// Struckig
// Copyright (C) 2022 Stefan Besler

// This program is free software: you can redistribute it and/or modify
// it under the terms of the GNU General Public License as published by
// the Free Software Foundation, either version 3 of the License, or
// (at your option) any later version.

// This program is distributed in the hope that it will be useful,
// but WITHOUT ANY WARRANTY; without even the implied warranty of
// MERCHANTABILITY or FITNESS FOR A PARTICULAR PURPOSE.  See the
// GNU General Public License for more details.
//
// You should have received a copy of the GNU General Public License
// along with THIS PROGRAM.  IF NOT, see <http://www.gnu.org/licenses/>.
/// Mathematical equations for Step 1 in third-order position interface: Extremal profiles
FUNCTION_BLOCK INTERNAL PositionThirdOrderStep1
VAR
  v0, a0 : LREAL;
  vf, af : LREAL;
  _vMax, _vMin, _aMax, _aMin, _jMax : LREAL;

  // Pre-calculated expressions
  pd : LREAL;
  v0_v0, vf_vf : LREAL;
  a0_a0, a0_p3, a0_p4 : LREAL;
  af_af, af_p3, af_p4 : LREAL;
  jMax_jMax : LREAL;
  
  // runtime  calculated expressions
  polynom_none, polynom_acc0, polynom_acc1 : ARRAY[0..4] OF LREAL;
  orig : LREAL;
  deriv : LREAL;
  t : LREAL;
  i : INT;
  h0, h1, h2, h2_h2, h3, h5, h2_none, h3_acc0, h3_acc1, h0_acc0, h2_acc0, h0_acc1, h2_acc1, q : LREAL;
  t_min, t_max, t_min_none, t_max_none, t_min_acc0, t_max_acc0, t_min_acc1, t_max_acc1 : LREAL;
  t_acc1, t_acc0 : LREAL;
  validProfiles : ARRAY[0..5] OF ProfileDesc; // Max 5 valid profiles + 1 spare for numerical issues
  validProfileCounter : INT := -1;
  
  num_roots_none, num_roots_acc0, num_roots_acc1  : INT;
  roots_none, roots_acc0, roots_acc1 : ARRAY[0..6] OF LREAL;
  roots_none_indices, roots_acc0_indices, roots_acc1_indices : ARRAY[0..6] OF INT;
  left_duration, right_duration : LREAL;   
END_VAR

METHOD AddInterval
VAR_IN_OUT
  interval : BlockInterval;
  Left : ProfileDesc;
  Right : ProfileDesc;
END_VAR
left_duration := Left.t_sum[6] + Left.Brake.Duration + Left.Accel.Duration;
right_duration := Right.t_sum[6] + Right.Brake.Duration + Right.Accel.Duration;
IF (left_duration < right_duration)
THEN
  interval.Left := left_duration;
  interval.Right := right_duration;
  interval.Profile := Right;
  interval.IsUsed := TRUE;
ELSE
  interval.Left := right_duration;
  interval.Right := left_duration;
  interval.Profile := Left;
  interval.IsUsed := TRUE;  
END_IF
END_METHOD

METHOD AddProfile
VAR_IN_OUT CONSTANT
  Profile : ProfileDesc;
END_VAR
validProfileCounter := validProfileCounter + 1;
validProfiles[validProfileCounter] := Profile;
END_METHOD

METHOD CalculateBlock : BOOL
VAR_IN_OUT
  block : Block;
END_VAR
VAR
  i, j : INT;
  Tmin : LREAL;
  idx_min : INT;
  idx_else_1, idx_else_2, idx_else_3, idx_else_4 : INT;
END_VAR
block.A.IsUsed := FALSE;
block.B.IsUsed := FALSE;

IF validProfileCounter = 0
THEN
  block.Pmin := validProfiles[0];
  block.Tmin := block.Pmin.t_sum[6] + block.Pmin.Brake.Duration + block.Pmin.Accel.Duration; 
  CalculateBlock := TRUE;

ELSIF validProfileCounter = 1 
THEN

  IF ABS(validProfiles[0].t_sum[6] - validProfiles[1].t_sum[6]) < 8*Constants.Epsilon
  THEN
    block.Pmin := validProfiles[0];
    block.Tmin := block.Pmin.t_sum[6] + block.Pmin.Brake.Duration + block.Pmin.Accel.Duration;  
    CalculateBlock := TRUE;
    RETURN;
	END_IF
  
  IF ParameterList.NumericalRobust
  THEN
    idx_min := SEL(validProfiles[0].t_sum[6] < validProfiles[1].t_sum[6], 1, 0);
    idx_else_1 := (idx_min + 1) MOD 2;

    block.Pmin := validProfiles[idx_min];
    block.Tmin := block.Pmin.t_sum[6] + block.Pmin.Brake.Duration + block.Pmin.Accel.Duration; 
    AddInterval(block.A, validProfiles[idx_min], validProfiles[idx_else_1]);
    CalculateBlock := TRUE;
    RETURN; 
	END_IF

// Only happens due to numerical issues
ELSIF (validProfileCounter = 3) 
THEN
  // Find "identical" profiles
  IF (ABS(validProfiles[0].t_sum[6] - validProfiles[1].t_sum[6]) < 32*Constants.Epsilon AND_THEN validProfiles[0].Direction <> validProfiles[1].Direction)
  THEN
    RemoveProfile(1);
  ELSIF (ABS(validProfiles[2].t_sum[6] - validProfiles[3].t_sum[6]) < 256*Constants.Epsilon  AND_THEN validProfiles[2].Direction <> validProfiles[3].Direction)
  THEN
    RemoveProfile(3);
  ELSIF (ABS(validProfiles[0].t_sum[6] - validProfiles[3].t_sum[6]) < 256*Constants.Epsilon AND_THEN validProfiles[0].Direction <> validProfiles[3].Direction)
  THEN
    RemoveProfile(3);
  ELSE
    RETURN;
  END_IF

ELSIF ((validProfileCounter+1) MOD 2 = 0)
THEN
  RETURN;
END_IF

// Find index of fastest Profile
Tmin := Constants.Infinity;
FOR i:=0 TO validProfileCounter
DO
  FOR j:=0 TO validProfileCounter
  DO
    IF validProfiles[i].t_sum[6] + validProfiles[i].Brake.Duration < validProfiles[j].t_sum[6] + validProfiles[j].Brake.Duration AND_THEN
       validProfiles[i].t_sum[6] + validProfiles[i].Brake.Duration < Tmin
    THEN
      Tmin := validProfiles[i].t_sum[6] + validProfiles[i].Brake.Duration + validProfiles[i].Accel.Duration;
      idx_min := i;
		END_IF
  END_FOR
END_FOR

block.Pmin := validProfiles[idx_min];
block.Tmin := block.Pmin.t_sum[6] + block.Pmin.Brake.Duration + block.Pmin.Accel.Duration;
IF (validProfileCounter = 2)
THEN
  idx_else_1 := (idx_min + 1) MOD 3;
  idx_else_2 := (idx_min + 2) MOD 3;
  
  AddInterval(block.A, validProfiles[idx_else_1], validProfiles[idx_else_2]);
  CalculateBlock := TRUE;
  RETURN;

 ELSIF (validProfileCounter = 4)
 THEN
  idx_else_1 := (idx_min + 1) MOD 5;
  idx_else_2 := (idx_min + 2) MOD 5;
  idx_else_3 := (idx_min + 3) MOD 5;
  idx_else_4 := (idx_min + 4) MOD 5;
  
  IF (validProfiles[idx_else_1].Direction = validProfiles[idx_else_2].Direction)
  THEN
    AddInterval(block.A, validProfiles[idx_else_1], validProfiles[idx_else_2]);
    AddInterval(block.B, validProfiles[idx_else_3], validProfiles[idx_else_4]);
  ELSE 
    AddInterval(block.A, validProfiles[idx_else_1], validProfiles[idx_else_4]);
    AddInterval(block.B, validProfiles[idx_else_2], validProfiles[idx_else_3]);
  END_IF
  
  CalculateBlock := TRUE;
END_IF
END_METHOD

METHOD Get : BOOL
VAR_INPUT
  input : REFERENCE TO ProfileDesc;
  block : REFERENCE TO Block; 
END_VAR
VAR_INST
  vMax, vMin, aMax, aMin, jMax : LREAL;  
END_VAR
validProfileCounter := -1;

// Zero-limits special case
IF _jMax = 0.0 OR_ELSE _aMax = 0.0 OR_ELSE _aMin = 0.0 
THEN
  block.Pmin.SetBoundary(input);

  IF time_all_single_step(block.Pmin, _vMax, _vMin, _aMax, _aMin, _jMax) 
  THEN
    block.Tmin := block.Pmin.t_sum[6] + block.Pmin.Brake.Duration + block.Pmin.Accel.Duration;
    AddInterval(block.A, block.Pmin, block.Pmin);
    
    IF ABS(v0) > Constants.DoubleEpsilon OR_ELSE ABS(a0) > Constants.DoubleEpsilon
    THEN
	  block.A.Left := block.Tmin;
      block.A.Right := Constants.Infinity;
    END_IF
    
    Get := TRUE;
    RETURN; 
  END_IF
  
  RETURN;
END_IF

validProfiles[0].SetBoundary(input);

IF ABS(vf) < Constants.DoubleEpsilon AND_THEN ABS(af) < Constants.DoubleEpsilon
THEN
  vMax := SEL(pd >= 0, _vMin, _vMax);
  vMin := SEL(pd >= 0, _vMax, _vMin);
  aMax := SEL(pd >= 0, _aMin, _aMax);
  aMin := SEL(pd >= 0, _aMax, _aMin);
  jMax :=SEL (pd >= 0,-_jMax, _jMax);
  
  IF ABS(v0) < Constants.DoubleEpsilon AND_THEN ABS(a0) < Constants.DoubleEpsilon AND_THEN ABS(pd) < Constants.DoubleEpsilon
  THEN
    time_all_none_acc0_acc1(input, vMax, vMin, aMax, aMin, jMax, TRUE);
  ELSE
    // There is no blocked interval when vf==0 && af==0, so return after first found profile
    time_all_vel(input, vMax, vMin, aMax, aMin, jMax, true);
    IF (validProfileCounter >= 0) THEN
      Get := CalculateBlock(block);
      RETURN;
    END_IF
    time_all_none_acc0_acc1(input, vMax, vMin, aMax, aMin, jMax, TRUE);
    IF (validProfileCounter >= 0) THEN
      Get := CalculateBlock(block);
      RETURN;
    END_IF
    time_acc0_acc1(input, vMax, vMin, aMax, aMin, jMax, true);
    IF (validProfileCounter >= 0) THEN
      Get := CalculateBlock(block);
      RETURN;
    END_IF
    
    time_all_vel(input, vMin, vMax, aMin, aMax, -jMax, true);
    IF (validProfileCounter >= 0) THEN
      Get := CalculateBlock(block);
      RETURN;
    END_IF
    time_all_none_acc0_acc1(input, vMin, vMax, aMin, aMax, -jMax, TRUE);
    IF (validProfileCounter >= 0) THEN
      Get := CalculateBlock(block);
      RETURN;
    END_IF
    time_acc0_acc1(input, vMin, vMax, aMin, aMax, -jMax, true);
  END_IF     

ELSE 
  time_all_none_acc0_acc1(input, _vMax, _vMin, _aMax, _aMin, _jMax, FALSE);
  time_all_none_acc0_acc1(input, _vMin, _vMax, _aMin, _aMax, -_jMax, false);
  time_acc0_acc1(input, _vMax, _vMin, _aMax, _aMin, _jMax, false);
  time_acc0_acc1(input, _vMin, _vMax, _aMin, _aMax, -_jMax, FALSE);
  time_all_vel(input, _vMax, _vMin, _aMax, _aMin, _jMax, FALSE);
  time_all_vel(input, _vMin, _vMax, _aMin, _aMax, -_jMax, false);  
END_IF    

IF (validProfileCounter = -1)
THEN
  time_none_two_step(input, _vMax, _vMin, _aMax, _aMin, _jMax);
  IF validProfileCounter >= 0
  THEN
    Get := CalculateBlock(block);
    RETURN;
	END_IF
  
  time_none_two_step(input, _vMin, _vMax, _aMin, _aMax, -_jMax);
  IF validProfileCounter >= 0
  THEN
    Get := CalculateBlock(block);
    RETURN;
	END_IF
  

  time_acc0_two_step(input, _vMax, _vMin, _aMax, _aMin, _jMax);
  IF validProfileCounter >= 0
  THEN
    Get := CalculateBlock(block);
    RETURN;
	END_IF
  
  time_acc0_two_step(input, _vMin, _vMax, _aMin, _aMax, -_jMax);
  IF validProfileCounter >= 0
  THEN
    Get := CalculateBlock(block);
    RETURN;
	END_IF
  
  time_vel_two_step(input, _vMax, _vMin, _aMax, _aMin, _jMax);
  IF validProfileCounter >= 0
  THEN
    Get := CalculateBlock(block);
    RETURN;
	END_IF
  
  time_vel_two_step(input, _vMin, _vMax, _aMin, _aMax, -_jMax);
  IF validProfileCounter >= 0
  THEN
    Get := CalculateBlock(block);
    RETURN;
	END_IF
  
  time_acc1_vel_two_step(input, _vMax, _vMin, _aMax, _aMin, _jMax);
  IF validProfileCounter >= 0
  THEN
    Get := CalculateBlock(block);
    RETURN;
	END_IF
  
  time_acc1_vel_two_step(input, _vMin, _vMax, _aMin, _aMax, -_jMax);
  IF validProfileCounter >= 0
  THEN
    Get := CalculateBlock(block);
    RETURN;
	END_IF  
END_IF

IF (validProfileCounter = -1)
THEN
  time_none_two_step(input, _vMax, _vMin, _aMax, _aMin, _jMax);
  IF validProfileCounter >= 0
  THEN
    Get := CalculateBlock(block);
    RETURN;
	END_IF
  
  time_none_two_step(input, _vMin, _vMax, _aMin, _aMax, -_jMax);
  IF validProfileCounter >= 0
  THEN
    Get := CalculateBlock(block);
    RETURN;
	END_IF
  

  time_acc0_two_step(input, _vMax, _vMin, _aMax, _aMin, _jMax);
  IF validProfileCounter >= 0
  THEN
    Get := CalculateBlock(block);
    RETURN;
	END_IF
  
  time_acc0_two_step(input, _vMin, _vMax, _aMin, _aMax, -_jMax);
  IF validProfileCounter >= 0
  THEN
    Get := CalculateBlock(block);
    RETURN;
	END_IF
  
  time_vel_two_step(input, _vMax, _vMin, _aMax, _aMin, _jMax);
  IF validProfileCounter >= 0
  THEN
    Get := CalculateBlock(block);
    RETURN;
	END_IF
  
  time_vel_two_step(input, _vMin, _vMax, _aMin, _aMax, -_jMax);
  IF validProfileCounter >= 0
  THEN
    Get := CalculateBlock(block);
    RETURN;
	END_IF
  
  time_acc1_vel_two_step(input, _vMax, _vMin, _aMax, _aMin, _jMax);
  IF validProfileCounter >= 0
  THEN
    Get := CalculateBlock(block);
    RETURN;
	END_IF
  
  time_acc1_vel_two_step(input, _vMin, _vMax, _aMin, _aMax, -_jMax);
  IF validProfileCounter >= 0
  THEN
    Get := CalculateBlock(block);
    RETURN;
	END_IF  
END_IF  

Get := CalculateBlock(block);
END_METHOD

METHOD PRIVATE RemoveProfile : BOOL
VAR_INPUT
  index : INT;
END_VAR
VAR
  i : INT;
END_VAR
// todo, this is pretty slow in twincat
FOR i:=index TO validProfileCounter-2
DO
  validProfiles[i] := validProfiles[i + 1];
END_FOR

validProfileCounter := validProfileCounter - 1;
END_METHOD

METHOD Set
VAR_INPUT
  p0, v0, a0 : LREAL;
  pf, vf, af : LREAL;
  vMax, vMin : LREAL;
  aMax, aMin : LREAL;
  jMax : LREAL;  
END_VAR
THIS^.v0 := v0;
THIS^.a0 := a0;
THIS^.vf := vf;
THIS^.af := af;
_vMax := vMax;
_vMin := vMin;
_aMax := aMax;
_aMin := aMin;
_jMax := jMax;

pd := pf - p0;

v0_v0 := v0 * v0;
vf_vf := vf * vf;

a0_a0 := a0 * a0;
af_af := af * af;

a0_p3 := a0 * a0_a0;
a0_p4 := a0_a0 * a0_a0;
af_p3 := af * af_af;
af_p4 := af_af * af_af;

// max values needs to be invariant to plus minus sign change
jMax_jMax := jMax * jMax;
END_METHOD

METHOD PRIVATE time_acc0_acc1
VAR_INPUT
  profile : REFERENCE TO ProfileDesc;
  vMax, vMin, aMax, aMin, jMax : LREAL;
  return_after_found : BOOL;  
END_VAR
h1 := (3*(af_p4*aMax - a0_p4*aMin) + aMax*aMin*(8*(a0_p3 - af_p3) + 3*aMax*aMin*(aMax - aMin) + 6*aMin*af_af - 6*aMax*a0_a0) + 12*jMax*(aMax*aMin*((aMax - 2*a0)*v0 - (aMin - 2*af)*vf) + aMin*a0_a0*v0 - aMax*af_af*vf))/(3*(aMax - aMin)*jMax_jMax) + 4*(aMax*vf_vf - aMin*v0_v0 - 2*aMin*aMax*pd)/(aMax - aMin);
IF (h1 >= 0) // check if h1 isNan
THEN
  h1 := SQRT(h1) * 0.5;
  h2 := a0_a0/(2*aMax*jMax) + (aMin - 2*aMax)/(2*jMax) - v0/aMax;
  h3 := -af_af/(2*aMin*jMax) - (aMax - 2*aMin)/(2*jMax) + vf/aMin;
  
  // UDDU: Solution 2
  IF h2 > h1/aMax AND_THEN h3 > -h1/aMin
  THEN
    profile.t[0] := (-a0 + aMax)/jMax;
    profile.t[1] := h2 - h1/aMax;
    profile.t[2] := aMax/jMax;
    profile.t[3] := 0;
    profile.t[4] := -aMin/jMax;
    profile.t[5] := h3 + h1/aMin;
    profile.t[6] := profile.t[4] + af/jMax;
  
    IF (profile.CheckVel(ProfileControlSigns.Uddu, ReachedLimits.Acc0Acc1, jMax, vMax, vMin, aMax, aMin, setLimits:=TRUE))
    THEN
      AddProfile(profile);
      IF return_after_found
      THEN
        RETURN;
			END_IF
    END_IF
  END_IF
  
  // UDDU: Solution 1  
  IF h2 > -h1/aMax AND_THEN h3 > h1/aMin
  THEN
    profile.t[0] := (-a0 + aMax)/jMax;
    profile.t[1] := h2 + h1/aMax;
    profile.t[2] := aMax/jMax;
    profile.t[3] := 0;
    profile.t[4] := -aMin/jMax;
    profile.t[5] := h3 - h1/aMin;
    profile.t[6] := profile.t[4] + af/jMax;
  
    IF (profile.CheckVel(ProfileControlSigns.Uddu, ReachedLimits.Acc0Acc1, jMax, vMax, vMin, aMax, aMin, setLimits:=TRUE))
    THEN
      AddProfile(profile);              
    END_IF
	END_IF  
END_IF
END_METHOD

/// Only for numerical issues, always return_after_found
METHOD PRIVATE time_acc0_two_step
VAR_INPUT
  profile : REFERENCE TO ProfileDesc;
  vMax, vMin, aMax, aMin, jMax : LREAL;
END_VAR
IF ABS(2*a0*jMax) > Constants.Epsilon
THEN
  // Two step
  profile.t[0] := 0;
  profile.t[1] := (af_af - a0_a0 + 2*jMax*(vf - v0))/(2*a0*jMax);
  profile.t[2] := (a0 - af)/jMax;
  profile.t[3] := 0;
  profile.t[4] := 0;
  profile.t[5] := 0;
  profile.t[6] := 0;
  
  IF (profile.CheckVel(ProfileControlSigns.Uddu, ReachedLimits.Acc0, jMax, vMax, vMin, aMax, aMin, setLimits:=FALSE))
  THEN
    AddProfile(profile);
    RETURN;
  END_IF
END_IF

// Three step - Removed pf
profile.t[0] := (-a0 + aMax)/jMax;
profile.t[1] := (a0_a0 + af_af - 2*aMax*aMax + 2*jMax*(vf - v0))/(2*aMax*jMax);
profile.t[2] := (-af + aMax)/jMax;
profile.t[3] := 0;
profile.t[4] := 0;
profile.t[5] := 0;
profile.t[6] := 0;

IF (profile.CheckVel(ProfileControlSigns.Uddu, ReachedLimits.Acc0, jMax, vMax, vMin, aMax, aMin, setLimits:=FALSE))
THEN
  AddProfile(profile);
  RETURN;     
END_IF


// Three step - Removed aMax
h0 := 3*(af_af - a0_a0 + 2*jMax*(v0 + vf));
h2 := a0_p3 + 2*af_p3 + 6*jMax_jMax*pd + 6*(af - a0)*jMax*vf - 3*a0*af_af;
h1 := 2*(2*h2*h2 + h0*(a0_p4 - 6*a0_a0*(af_af + 2*jMax*vf) + 8*a0*(af_p3 + 3*jMax_jMax*pd + 3*af*jMax*vf) - 3*(af_p4 + 4*af_af*jMax*vf + 4*jMax_jMax*(vf_vf - v0_v0))));
IF h1 >= 0 AND_THEN ABS(h0) > Constants.DoubleEpsilon
THEN
  h1 := SQRT(h1) * ABS(jMax) / jMax;
  
  profile.t[0] := (4*af_p3 + 2*a0_p3 - 6*a0*af_af + 12*jMax_jMax*pd + 12*(af - a0)*jMax*vf + h1)/(2*jMax*h0);
  profile.t[1] := -h1/(jMax*h0);
  profile.t[2] := (-4*a0_p3 - 2*af_p3 + 6*a0_a0*af + 12*jMax_jMax*pd - 12*(af - a0)*jMax*v0 + h1)/(2*jMax*h0);
  profile.t[3] := 0;
  profile.t[4] := 0;
  profile.t[5] := 0;
  profile.t[6] := 0;
  
  IF (profile.CheckVel(ProfileControlSigns.Uddu, ReachedLimits.Acc0, jMax, vMax, vMin, aMax, aMin, setLimits:=FALSE))
  THEN
    AddProfile(profile);
    RETURN;     
  END_IF
END_IF


// Three step - t=(aMax - aMin)/jMax
t := (aMax - aMin)/jMax;

profile.t[0] := (-a0 + aMax)/jMax;
profile.t[1] := (a0_a0 - af_af)/(2*aMax*jMax) + (vf - v0 + jMax*t*t)/aMax - 2*t;
profile.t[2] := t;
profile.t[3] := 0;
profile.t[4] := 0;
profile.t[5] := 0;
profile.t[6] := (af - aMin)/jMax;

IF (profile.CheckVel(ProfileControlSigns.Uddu, ReachedLimits.Acc0, jMax, vMax, vMin, aMax, aMin, setLimits:=FALSE))
THEN
  AddProfile(profile);
  RETURN;     
END_IF
END_METHOD

/// Only for numerical issues, always return_after_found
METHOD PRIVATE time_acc1_vel_two_step
VAR_INPUT
  profile : REFERENCE TO ProfileDesc;
  vMax, vMin, aMax, aMin, jMax : LREAL;
END_VAR

IF ABS(vMax) < Constants.DoubleEpsilon
THEN
  RETURN;
END_IF

profile.t[0] := 0;
profile.t[1] := 0;
profile.t[2] := a0/jMax;
profile.t[3] := -(3*af_p4 - 8*aMin*(af_p3 - a0_p3) - 24*aMin*jMax*(a0*v0 - af*vf) + 6*af_af*(aMin*aMin - 2*jMax*vf) - 12*jMax*(2*aMin*jMax*pd + aMin*aMin*(vf + vMax) + jMax*(vMax*vMax - vf_vf) + aMin*a0*(a0_a0 - 2*jMax*(v0 + vMax))/jMax))/(24*aMin*jMax_jMax*vMax);
profile.t[4] := -aMin/jMax;
profile.t[5] := -(af_af/2 - aMin*aMin + jMax*(vMax - vf))/(aMin*jMax);
profile.t[6] := profile.t[4] + af/jMax;

IF (Profile.CheckVel(ProfileControlSigns.Uddu, ReachedLimits.Acc1Vel, jMax, vMax, vMin, aMax, aMin, setLimits:=FALSE))
THEN
  AddProfile(Profile);
  RETURN;        
END_IF
END_METHOD

METHOD PRIVATE time_all_none_acc0_acc1
VAR_INPUT
  profile : REFERENCE TO ProfileDesc;
  vMax, vMin, aMax, aMin, jMax : LREAL;
  return_after_found : BOOL;
END_VAR
// NONE UDDU / UDUD Strategy: t7 == 0 (equals UDDU), this one is in particular prone to numerical issues
h2_none := (a0_a0 - af_af)/(2*jMax) + (vf - v0);
h2_h2 := h2_none*h2_none;
t_min_none := (a0 - af)/jMax;
t_max_none := (aMax - aMin)/jMax;

polynom_none[0] := 0;
polynom_none[1] := -2*(a0_a0 + af_af - 2*jMax*(v0 + vf))/jMax_jMax;
polynom_none[2] := 4*(a0_p3 - af_p3 + 3*jMax*(af*vf - a0*v0))/(3*jMax*jMax_jMax) - 4*pd/jMax;
polynom_none[3] := -h2_h2/jMax_jMax;

// ACC0
h3_acc0 := (a0_a0 - af_af)/(2*aMax*jMax) + (vf - v0)/aMax;
t_min_acc0 := (aMax - af)/jMax;
t_max_acc0 := (aMax - aMin)/jMax;

h0_acc0 := 3*(af_p4 - a0_p4) + 8*(a0_p3 - af_p3)*aMax + 24*aMax*jMax*(af*vf - a0*v0) - 6*a0_a0*(aMax*aMax - 2*jMax*v0) + 6*af_af*(aMax*aMax - 2*jMax*vf) + 12*jMax*(jMax*(vf_vf - v0_v0 - 2*aMax*pd) - aMax*aMax*(vf - v0));
h2_acc0 := -af_af + aMax*aMax + 2*jMax*vf;

polynom_acc0[0] := -2*aMax/jMax;
polynom_acc0[1] := h2_acc0/jMax_jMax;
polynom_acc0[2] := 0;
polynom_acc0[3] := h0_acc0/(12*jMax_jMax*jMax_jMax);

// ACC1
h3_acc1 := -(a0_a0 + af_af)/(2*jMax*aMin) + aMin/jMax + (vf - v0)/aMin;
t_min_acc1 := (aMin - a0)/jMax;
t_max_acc1 := (aMax - a0)/jMax;

h0_acc1 := (a0_p4 - af_p4)/4 + 2*(af_p3 - a0_p3)*aMin/3 + (a0_a0 - af_af)*aMin*aMin/2 + jMax*(af_af*vf + a0_a0*v0 + 2*aMin*(jMax*pd - a0*v0 - af*vf) + aMin*aMin*(v0 + vf) + jMax*(v0_v0 - vf_vf));
h2_acc1 := a0_a0 - a0*aMin + 2*jMax*v0;

polynom_acc1[0] := 2*(2*a0 - aMin)/jMax;
polynom_acc1[1] := (5*a0_a0 + aMin*(aMin - 6*a0) + 2*jMax*v0)/jMax_jMax;
polynom_acc1[2] := 2*(a0 - aMin)*h2_acc1/(jMax_jMax*jMax);
polynom_acc1[3] := h0_acc1/(jMax_jMax*jMax_jMax);

Roots.SolveQuartMonic(ADR(polynom_none), 4, rootCount:=num_roots_none, roots:=roots_none);
Roots.SolveQuartMonic(ADR(polynom_acc0), 4, rootCount:=num_roots_acc0, roots:=roots_acc0);
Roots.SolveQuartMonic(ADR(polynom_acc1), 4, rootCount:=num_roots_acc1, roots:=roots_acc1);

BubbleSortLreal(ADR(roots_none), num_roots_none, ADR(roots_none_indices));
BubbleSortLreal(ADR(polynom_acc0), num_roots_acc0, ADR(roots_acc0_indices));
BubbleSortLreal(ADR(polynom_acc1), num_roots_acc1, ADR(roots_acc1_indices));

FOR i:=0 TO num_roots_none
DO
  t := roots_none[roots_none_indices[i]];
  IF t < t_min_none OR_ELSE t > t_max_none
  THEN
    CONTINUE;
	END_IF
            
  // Single Newton-step (regarding pd)
  IF (t > Constants.DoubleEpsilon)
  THEN
    h1 := jMax*t*t;
    orig := -h2_h2/(4*jMax*t) + h2_none*(af/jMax + t) + (4*a0_p3 + 2*af_p3 - 6*a0_a0*(af + 2*jMax*t) + 12*(af - a0)*jMax*v0 + 3*jMax_jMax*(-4*pd + (h1 + 8*v0)*t))/(12*jMax_jMax);
    deriv := h2_none + 2*v0 - a0_a0/jMax + h2_h2/(4*h1) + (3*h1)/4;
    IF ABS(deriv) < Constants.DoubleEpsilon
    THEN
      CONTINUE;
    END_IF
    
    t := t - orig / deriv;
  END_IF
  
  IF (t <= Constants.DoubleEpsilon)
  THEN
    CONTINUE;
  END_IF
  
  h0 := h2_none/(2*jMax*t);
  profile.t[0] := h0 + t/2 - a0/jMax;
  profile.t[1] := 0;
  profile.t[2] := t;
  profile.t[3] := 0;
  profile.t[4] := 0;
  profile.t[5] := 0;
  profile.t[6] := -h0 + t/2 + af/jMax;

  IF (profile.CheckVel(ProfileControlSigns.Uddu, ReachedLimits.None, jMax, vMax, vMin, aMax, aMin, setLimits:=FALSE)) 
  THEN
    AddProfile(profile);
    IF return_after_found
    THEN
      RETURN;
		END_IF
  END_IF
END_FOR     
    
FOR i:=0 TO num_roots_acc0
DO
  t := roots_acc0[roots_acc0_indices[i]];
  IF t < t_min_acc0 OR_ELSE t > t_max_acc0
  THEN
    CONTINUE;
  END_IF
  
  // Single Newton step (regarding pd)
  IF t > Constants.DoubleEpsilon
  THEN
    h1 := jMax*t;
    orig := h0_acc0/(12*jMax_jMax*t) + t*(h2_acc0 + h1*(h1 - 2*aMax));
    deriv := 2*(h2_acc0 + h1*(2*h1 - 3*aMax));
    IF ABS(deriv) > Constants.DoubleEpsilon
    THEN
      t := t - orig / deriv;
    END_IF
  END_IF
  
  IF ABS(deriv) < Constants.DoubleEpsilon
  THEN
    CONTINUE;
	END_IF
  
  profile.t[0] := (-a0 + aMax)/jMax;
  profile.t[1] := h3_acc0 - 2*t + jMax/aMax*t*t;
  profile.t[2] := t;
  profile.t[3] := 0;
  profile.t[4] := 0;
  profile.t[5] := 0;
  profile.t[6] := (af - aMax)/jMax + t;
  
  IF (profile.CheckVel(ProfileControlSigns.Uddu, ReachedLimits.Acc0, jMax, vMax, vMin, aMax, aMin, setLimits:=FALSE))
  THEN
    AddProfile(profile);
    IF return_after_found
    THEN
      RETURN;
		END_IF    
  END_IF
END_FOR

FOR i:=0 TO num_roots_acc1
DO
  t := roots_acc1[roots_acc1_indices[i]];
  IF t < t_min_acc1 OR_ELSE t > t_max_acc1 THEN
    CONTINUE;
  END_IF 

  IF t > Constants.DoubleEpsilon
  THEN
    // Double Newton step (regarding pd)
    h5 := a0_p3 + 2*jMax*a0*v0;
    h1 := jMax*t;
    orig := -(h0_acc1/2 + h1*(h5 + a0*(aMin - 2*h1)*(aMin - h1) + a0_a0*(5*h1/2 - 2*aMin) + aMin*aMin*h1/2 + jMax*(h1/2 - aMin)*(h1*t + 2*v0)))/jMax;
    deriv := (aMin - a0 - h1)*(h2_acc1 + h1*(4*a0 - aMin + 2*h1));
    IF ABS(deriv) > Constants.DoubleEpsilon
    THEN
      t := t - MIN(orig / deriv, t);
      
      h1 := jMax*t;
      orig := -(h0_acc1/2 + h1*(h5 + a0*(aMin - 2*h1)*(aMin - h1) + a0_a0*(5*h1/2 - 2*aMin) + aMin*aMin*h1/2 + jMax*(h1/2 - aMin)*(h1*t + 2*v0)))/jMax;
      IF (ABS(orig) > 1E-9)
      THEN
        deriv := (aMin - a0 - h1)*(h2_acc1 + h1*(4*a0 - aMin + 2*h1));
        
        IF ABS(deriv) > Constants.DoubleEpsilon
        THEN
          t := t - orig / deriv; 
          h1 := jMax*t;
          orig := -(h0_acc1/2 + h1*(h5 + a0*(aMin - 2*h1)*(aMin - h1) + a0_a0*(5*h1/2 - 2*aMin) + aMin*aMin*h1/2 + jMax*(h1/2 - aMin)*(h1*t + 2*v0)))/jMax;

          IF ABS(orig) > 1E-9
          THEN
            deriv := (aMin - a0 - h1)*(h2_acc1 + h1*(4*a0 - aMin + 2*h1));
            
            IF ABS(deriv) > Constants.DoubleEpsilon
            THEN            
              t := t -orig / deriv;
            END_IF
          END_IF
        END_IF
      END_IF 
    END_IF  
	END_IF

  profile.t[0] := t;
  profile.t[1] := 0;
  profile.t[2] := (a0 - aMin)/jMax + t;
  profile.t[3] := 0;
  profile.t[4] := 0;
  profile.t[5] := h3_acc1 - (2*a0 + jMax*t)*t/aMin;
  profile.t[6] := (af - aMin)/jMax;
  
  IF (profile.CheckVel(ProfileControlSigns.Uddu, ReachedLimits.Acc1, jMax, vMax, vMin, aMax, aMin, setLimits:=TRUE))
  THEN
    AddProfile(profile);
    IF return_after_found
    THEN
      RETURN;
		END_IF    
  END_IF
END_FOR
END_METHOD

METHOD PRIVATE time_all_single_step : BOOL
VAR_INPUT
  profile : REFERENCE TO ProfileDesc;
  vMax, vMin, aMax, aMin, jMax : LREAL;
END_VAR
IF ABS(af - a0) > Constants.DoubleEpsilon
THEN
  RETURN;
END_IF

profile.t[0] := 0;
profile.t[1] := 0;
profile.t[2] := 0;
profile.t[3] := 0;
profile.t[4] := 0;
profile.t[5] := 0;
profile.t[6] := 0;

IF ABS(a0) > Constants.DoubleEpsilon
THEN
  q := 2*a0*pd + v0_v0;
  IF q >= 0
  THEN
    q := SQRT(q);
    
    // Solution 1
    profile.t[3] := (-v0 + q) / a0;
    IF profile.t[3] >= 0.0 AND_THEN profile.CheckVel(ProfileControlSigns.Uddu, ReachedLimits.None, 0.0, vMax, vMin, aMax, aMin, FALSE)
    THEN
      AddProfile(profile);
      time_all_single_step := TRUE;
      RETURN;
    END_IF  
    
    // Solution 2
    profile.t[3] := -(v0 + q) / a0;
    IF profile.CheckVel(ProfileControlSigns.Uddu, ReachedLimits.None, 0.0, vMax, vMin, aMax, aMin, FALSE)
    THEN
      AddProfile(profile);
      time_all_single_step := TRUE;
      RETURN;
    END_IF
  END_IF
  
ELSIF ABS(v0) > Constants.DoubleEpsilon
THEN
  profile.t[3] := pd / v0;
  IF profile.CheckVel(ProfileControlSigns.Uddu, ReachedLimits.None, 0.0, vMax, vMin, aMax, aMin, FALSE)
  THEN
    time_all_single_step := TRUE;
    RETURN;
  END_IF
  
ELSIF ABS(pd) < Constants.DoubleEpsilon
THEN 
  IF profile.CheckVel(ProfileControlSigns.Uddu, ReachedLimits.None, 0.0, vMax, vMin, aMax, aMin, FALSE)
  THEN
    time_all_single_step := TRUE;
    RETURN;
  END_IF      
END_IF
END_METHOD

METHOD PRIVATE time_all_vel
VAR_INPUT
  profile : REFERENCE TO ProfileDesc;
  vMax, vMin, aMax, aMin, jMax : LREAL;
  return_after_found : BOOL;  
END_VAR

IF ABS(vMax) < Constants.DoubleEpsilon
THEN
  RETURN;
END_IF

// ACC0_ACC1_VEL
profile.t[0] := (-a0 + aMax)/jMax;
profile.t[1] := (a0_a0*0.5 - aMax*aMax - jMax*(v0 - vMax))/(aMax*jMax);
profile.t[2] := aMax/jMax;
profile.t[3] := (3*(a0_p4*aMin - af_p4*aMax) + 8*aMax*aMin*(af_p3 - a0_p3 + 3*jMax*(a0*v0 - af*vf)) + 6*a0_a0*aMin*(aMax*aMax - 2*jMax*v0) - 6*af_af*aMax*(aMin*aMin - 2*jMax*vf) - 12*jMax*(aMax*aMin*(aMax*(v0 + vMax) - aMin*(vf + vMax) - 2*jMax*pd) + (aMin - aMax)*jMax*vMax*vMax + jMax*(aMax*vf_vf - aMin*v0_v0)))/(24*aMax*aMin*jMax_jMax*vMax);
profile.t[4] := -aMin/jMax;
profile.t[5] := -(af_af*0.5 - aMin*aMin - jMax*(vf - vMax))/(aMin*jMax);
profile.t[6] := profile.t[4] + af/jMax;

IF (profile.CheckVel(ProfileControlSigns.Uddu, ReachedLimits.Acc0Acc1Vel, jMax, vMax, vMin, aMax, aMin, setLimits:=FALSE))
THEN
  AddProfile(profile);
  RETURN;    
END_IF

// ACC1_VEL
t_acc0  := a0_a0/(2*jMax_jMax) + (vMax - v0)/jMax;
IF t_acc0 >= 0
THEN
  t_acc0 := SQRT(t_acc0 );
  profile.t[0] := t_acc0  - a0/jMax;
  profile.t[1] := 0;
  profile.t[2] := t_acc0 ;
  profile.t[3] := -(3*af_p4 - 8*aMin*(af_p3 - a0_p3) - 24*aMin*jMax*(a0*v0 - af*vf) + 6*af_af*(aMin*aMin - 2*jMax*vf) - 12*jMax*(2*aMin*jMax*pd + aMin*aMin*(vf + vMax) + jMax*(vMax*vMax - vf_vf) + aMin*t_acc0 *(a0_a0 - 2*jMax*(v0 + vMax))))/(24*aMin*jMax_jMax*vMax);
  //profile.t[4] := -aMin/jMax;
  //profile.t[5] := -(af_af*0.5 - aMin*aMin + jMax*(vMax - vf))/(aMin*jMax);
  //profile.t[6] := profile.t[4] + af/jMax;
        
  IF (profile.CheckVel(ProfileControlSigns.Uddu, ReachedLimits.Acc1Vel, jMax, vMax, vMin, aMax, aMin, setLimits:=FALSE)) 
  THEN
    AddProfile(profile); 
    RETURN; 
  END_IF
END_IF

// ACC0_VEL
t_acc1 := 0.5*af_af/(jMax_jMax) + (vMax - vf)/jMax;
IF t_acc1 >= 0
THEN
  t_acc1 := SQRT(t_acc1);
  profile.t[0] := (-a0 + aMax)/jMax;
  profile.t[1] := (a0_a0*0.5 - aMax*aMax - jMax*(v0 - vMax))/(aMax*jMax);
  profile.t[2] := aMax/jMax;
  profile.t[3] := (3*a0_p4 + 8*aMax*(af_p3 - a0_p3) + 24*aMax*jMax*(a0*v0 - af*vf) + 6*a0_a0*(aMax*aMax - 2*jMax*v0) - 12*jMax*(-2*aMax*jMax*pd + aMax*aMax*(v0 + vMax) + jMax*(vMax*vMax - v0_v0) + aMax*t_acc1*(-af_af + 2*(vf + vMax)*jMax)))/(24*aMax*jMax_jMax*vMax);
  profile.t[4] := t_acc1;
  profile.t[5] := 0;
  profile.t[6] := t_acc1 + af/jMax;
  
  IF (profile.CheckVel(ProfileControlSigns.Uddu, ReachedLimits.Acc0Vel, jMax, vMax, vMin, aMax, aMin, setLimits:=FALSE)) 
  THEN
    AddProfile(profile);
    RETURN;
  END_IF
END_IF

// VEL
// Solution 3/4
IF t_acc0 >= 0 AND_THEN t_acc1 >= 0
THEN
  profile.t[0] := t_acc0 - a0/jMax;
  profile.t[1] := 0;
  profile.t[2] := t_acc0;
  profile.t[3] := (af_p3 - a0_p3)/(3.0*jMax_jMax*vMax) + (a0*v0 - af*vf + (af_af*t_acc1 + a0_a0*t_acc0)*0.5)/(jMax*vMax) - (v0/vMax + 1.0)*t_acc0 - (vf/vMax + 1.0)*t_acc1 + pd/vMax;
  //profile.t[4] := t_acc1;
  //profile.t[5] := 0;
  //profile.t[6] := t_acc1 + af/jMax;
  
  IF (profile.CheckVel(ProfileControlSigns.Uddu, ReachedLimits.Vel, jMax, vMax, vMin, aMax, aMin, setLimits:=FALSE))
  THEN
    AddProfile(profile);
    RETURN;
  END_IF
END_IF
END_METHOD

/// Only for numerical issues, always return_after_found
METHOD PRIVATE time_none_two_step
VAR_INPUT
  profile : REFERENCE TO ProfileDesc;
  vMax, vMin, aMax, aMin, jMax : LREAL;
END_VAR
// Two step
{}
  h0 := (a0_a0 + af_af)/2 + jMax*(vf - v0);
  IF h0 >= 0
  THEN
    h0 := SQRT(h0) * ABS(jMax) / jMax;
    profile.t[0] := (h0 - a0)/jMax;
    profile.t[1] := 0;
    profile.t[2] := (h0 - af)/jMax;
    profile.t[3] := 0;
    profile.t[4] := 0;
    profile.t[5] := 0;
    profile.t[6] := 0;
    
    IF (profile.CheckVel(ProfileControlSigns.Uddu, ReachedLimits.None, jMax, vMax, vMin, aMax, aMin, setLimits:=FALSE))
    THEN 
      AddProfile(profile);
      RETURN;
    END_IF
	END_IF
{}
  
  // Single step
{}
  profile.t[0] := (af - a0)/jMax;
  profile.t[1] := 0;
  profile.t[2] := 0;
  profile.t[3] := 0;
  profile.t[4] := 0;
  profile.t[5] := 0;
  profile.t[6] := 0;
  
  IF (profile.CheckVel(ProfileControlSigns.Uddu, ReachedLimits.None, jMax, vMax, vMin, aMax, aMin, setLimits:=FALSE))
  THEN 
    AddProfile(profile);
    RETURN;
  END_IF
{}
END_METHOD

/// Only for numerical issues, always return_after_found
METHOD PRIVATE time_vel_two_step
VAR_INPUT
  profile : REFERENCE TO ProfileDesc;
  vMax, vMin, aMax, aMin, jMax : LREAL;
END_VAR
h1 := af_af/(2*jMax_jMax) + (vMax - vf)/jMax;

IF h1 >= 0 AND_THEN ABS(vMax) > Constants.DoubleEpsilon
THEN
  h1 := SQRT(h1);
  
  // Four step
  {}    
    // Solution 3/4
    profile.t[0] := -a0/jMax;
    profile.t[1] := 0;
    profile.t[2] := 0;
    profile.t[3] := (af_p3 - a0_p3)/(3*jMax_jMax*vMax) + (a0*v0 - af*vf + (af_af*h1)/2)/(jMax*vMax) - (vf/vMax + 1.0)*h1 + pd/vMax;
    profile.t[4] := h1;
    profile.t[5] := 0;
    profile.t[6] := h1 + af/jMax;
  
    IF profile.CheckVel(ProfileControlSigns.Uddu, ReachedLimits.Vel, jMax, vMax, vMin, aMax, aMin, setLimits:=FALSE)
    THEN
      AddProfile(profile);
      RETURN;
    END_IF 
  {}
  
  {}    
    // Four step        
    profile.t[0] := 0;
    profile.t[1] := 0;
    profile.t[2] := a0/jMax;
    profile.t[3] := (af_p3 - a0_p3)/(3.0*jMax_jMax*vMax) + (a0*v0 - af*vf + (af_af*h1 + a0_p3/jMax)*0.5)/(jMax*vMax) - (v0/vMax + 1.0)*a0/jMax - (vf/vMax + 1.0)*h1 + pd/vMax;
    profile.t[4] := h1;
    profile.t[5] := 0;
    profile.t[6] := h1 + af/jMax;
    
    IF (profile.CheckVel(ProfileControlSigns.Uddu, ReachedLimits.Vel, jMax, vMax, vMin, aMax, aMin, setLimits:=FALSE))
    THEN
      AddProfile(profile); 
      RETURN;       
    END_IF
  {}
END_IF
END_METHOD

END_FUNCTION_BLOCK

(* stored: Version 1.1.0.1
   POU PositionThirdOrderStep1: Id {59242074-56b3-4cce-98f4-96108527bef2}, SpecialFunc None
   Method AddInterval: Id {f04cf183-f22e-4a08-854f-8d9fd235e3cd}
   Method AddProfile: Id {443ac9a1-c2c8-4422-873c-d80f090e8e87}
   Method CalculateBlock: Id {50e177a8-dca6-48ec-aabe-f9c22fb4f02a}
   Method Get: Id {1c1bdad0-f955-4d7e-82c0-f0b69b7c5251}
   Method RemoveProfile: Id {bd3a75f9-6643-430d-baa6-3b74a1498442}
   Method Set: Id {ce744db4-d360-45a6-a3e4-2c7d816397cb}
   Method time_acc0_acc1: Id {e5212c06-396a-492c-bc44-27957c4ab5ed}
   Method time_acc0_two_step: Id {bb72dd1e-fc6d-4110-a222-a9ef280818c2}
   Method time_acc1_vel_two_step: Id {64e54b1d-928d-4828-9fe0-4384e30cc74c}
   Method time_all_none_acc0_acc1: Id {05662139-7683-4090-a8b9-92a5e7494597}
   Method time_all_single_step: Id {55ad35e0-a00f-4e02-8b7d-a7106d66f7c6}
   Method time_all_vel: Id {0932514e-6750-4a1f-b673-619a59e1903e}
   Method time_none_two_step: Id {6056e359-3c2c-4ebb-b6ec-b0674ae1ae17}
   Method time_vel_two_step: Id {78d50b14-2a01-494d-b78f-ace6c4afe469} *)
